Fanuc TP program (LS listing): UP022.LS

/PROG  UP022
/ATTR
OWNER		= MNEDITOR;
COMMENT		= "Soldadura Est.";
PROG_SIZE	= 11568;
CREATE		= DATE 23-07-08  TIME 22:50:50;
MODIFIED	= DATE 24-03-09  TIME 08:24:52;
FILE_NAME	= UP002;
VERSION		= 0;
LINE_COUNT	= 53;
MEMORY_SIZE	= 20152;
PROTECT		= READ_WRITE;
TCD:  STACK_SIZE	= 500,
      TASK_PRIORITY	= 50,
      TIME_SLICE	= 0,
      BUSY_LAMP_OFF	= 0,
      ABORT_REQUEST	= 0,
      PAUSE_REQUEST	= 0;
DEFAULT_GROUP	= 1,1,1,1,*;
CONTROL_CODE	= 00000001 00000000;
/APPL
/MN
   1:  UFRAME_NUM=1 ;
   2:  UTOOL_NUM=2 ;
   3:  PAYLOAD[2] ;
   4:J P[1] 100% CNT0 ACC100 TB    .10sec,P-SPS    ;
      1:  TC_ONLINE (ON) ;
      2:  DO[23]=OFF ;
      3:  TIMER[4]=RESET ;
      4:  TIMER[4]=START ;
      5:  CALL MAKRO050    ;
      6:  !Lib. de Herramientas ;
      7:  DO[80]=ON ;
      8:  DO[78]=OFF ;
      9:  DO[77]=ON ;
     10:  DO[75]=OFF ;
     11:  !Lib. de Anticolisiones ;
     12:  DO[41]=ON ;
     13:  DO[42]=ON ;
     14:  DO[43]=ON ;
     15:  DO[44]=ON ;
     16:  !Apagar Pos. Base ;
     17:  DO[15]=OFF ;
     18:  !Robot en Trayectoria ;
     19:  DO[16]=ON ;
     20:  !Basculante 1 en Pos. de Reposo ;
     21:  IF (!DI[842] AND DO[12]),CALL MAKRO072 ;
     22:  WAIT (M[96])    ;
     23:  WAIT (DI[23])    ;
     24:  DO[23]=(ON) ;
     25:  TC_ONLINE (M[1] AND M[30] AND M[31] AND M[34] AND M[35] AND M[95] AND M[96]) ;
       ------ ;
   5:J P[2] 100% CNT100 ACC100 TB   0.00sec,P-SPS    ;
      1:  TC_ONLINE (M[1] AND M[30] AND M[31] AND M[34] AND M[35] AND M[95] AND M[96]) ;
       ------ ;
   6:J P[3] 100% CNT100 ACC100 TB   0.00sec,P-SPS    ;
      1:  TC_ONLINE (M[1] AND M[30] AND M[31] AND M[34] AND M[35] AND M[95] AND M[96]) ;
       ------ ;
   7:J P[4] 100% CNT100 ACC100 TB   0.00sec,P-SPS    ;
      1:  TC_ONLINE (M[1] AND M[30] AND M[31] AND M[34] AND M[35] AND M[95] AND M[96]) ;
       ------ ;
   8:  !5QA802035b_017_R_PS_0031 ;
   9:  !Punto de Sol. No. 10094 ;
  10:J P[5] 100% CNT0 ACC100 TB    .10sec,P-SPS Offset,PR[11]    ;
      1:  TC_ONLINE (ON) ;
      2:  DO[23]=OFF ;
      3:  WAIT (!DI[16] AND DI[23])    ;
      4:  CALL VW_USER(Basic1,EZSP,Nr1,ProgNr=99, , ,S-Punkt=10094,Fzg_Typ=7,EIN/AUS=ON) ;
      5:  GO[2]=(R[197]) ;
      6:  WAIT (!DI[129] OR DI[26])    ;
      7:  CALL MAKRO080    ;
      8:  WAIT (DI[23])    ;
      9:  DO[23]=ON ;
     10:  TC_ONLINE (M[1] AND M[30] AND M[31] AND M[34] AND M[35] AND M[95] AND M[96]) ;
       ------ ;
  11:  !5QA802035b_017_R_PS_0029 ;
  12:  !Punto de Sol. No. 10095 ;
  13:J P[6] 100% CNT0 ACC100 TB    .10sec,P-SPS Offset,PR[11]    ;
      1:  TC_ONLINE (ON) ;
      2:  DO[23]=OFF ;
      3:  WAIT (!DI[16] AND DI[23])    ;
      4:  CALL VW_USER(Basic1,EZSP,Nr1,ProgNr=99, , ,S-Punkt=10095,Fzg_Typ=7,EIN/AUS=ON) ;
      5:  GO[2]=(R[197]) ;
      6:  WAIT (!DI[129] OR DI[26])    ;
      7:  CALL MAKRO080    ;
      8:  WAIT (DI[23])    ;
      9:  DO[23]=ON ;
     10:  TC_ONLINE (M[1] AND M[30] AND M[31] AND M[34] AND M[35] AND M[95] AND M[96]) ;
       ------ ;
  14:  !5QA802035b_017_R_PS_0028 ;
  15:  !Punto de Sol. No. 10096 ;
  16:J P[7] 100% CNT0 ACC100 TB    .10sec,P-SPS Offset,PR[11]    ;
      1:  TC_ONLINE (ON) ;
      2:  DO[23]=OFF ;
      3:  WAIT (!DI[16] AND DI[23])    ;
      4:  CALL VW_USER(Basic1,EZSP,Nr1,ProgNr=99, , ,S-Punkt=10096,Fzg_Typ=7,EIN/AUS=ON) ;
      5:  GO[2]=(R[197]) ;
      6:  WAIT (!DI[129] OR DI[26])    ;
      7:  CALL MAKRO080    ;
      8:  WAIT (DI[23])    ;
      9:  DO[23]=ON ;
     10:  TC_ONLINE (M[1] AND M[30] AND M[31] AND M[34] AND M[35] AND M[95] AND M[96]) ;
       ------ ;
  17:  !5QA802035b_017_R_PS_0027 ;
  18:  !Punto de Sol. No. 10097 ;
  19:J P[8] 100% CNT0 ACC100 TB    .10sec,P-SPS Offset,PR[11]    ;
      1:  TC_ONLINE (ON) ;
      2:  DO[23]=OFF ;
      3:  WAIT (!DI[16] AND DI[23])    ;
      4:  CALL VW_USER(Basic1,EZSP,Nr1,ProgNr=99, , ,S-Punkt=10097,Fzg_Typ=7,EIN/AUS=ON) ;
      5:  GO[2]=(R[197]) ;
      6:  WAIT (!DI[129] OR DI[26])    ;
      7:  CALL MAKRO080    ;
      8:  WAIT (DI[23])    ;
      9:  DO[23]=ON ;
     10:  TC_ONLINE (M[1] AND M[30] AND M[31] AND M[34] AND M[35] AND M[95] AND M[96]) ;
       ------ ;
  20:  !5QA802035b_017_R_PS_0026 ;
  21:  !Punto de Sol. No. 10098 ;
  22:J P[9] 100% CNT0 ACC100 TB    .10sec,P-SPS Offset,PR[11]    ;
      1:  TC_ONLINE (ON) ;
      2:  DO[23]=OFF ;
      3:  WAIT (!DI[16] AND DI[23])    ;
      4:  CALL VW_USER(Basic1,EZSP,Nr1,ProgNr=99, , ,S-Punkt=10098,Fzg_Typ=7,EIN/AUS=ON) ;
      5:  GO[2]=(R[197]) ;
      6:  WAIT (!DI[129] OR DI[26])    ;
      7:  CALL MAKRO080    ;
      8:  WAIT (DI[23])    ;
      9:  DO[23]=ON ;
     10:  TC_ONLINE (M[1] AND M[30] AND M[31] AND M[34] AND M[35] AND M[95] AND M[96]) ;
       ------ ;
  23:  !5QA802035b_017_R_PS_0025 ;
  24:  !Punto de Sol. No. 10099 ;
  25:J P[10] 100% CNT0 ACC100 TB    .10sec,P-SPS Offset,PR[11]    ;
      1:  TC_ONLINE (ON) ;
      2:  DO[23]=OFF ;
      3:  WAIT (!DI[16] AND DI[23])    ;
      4:  CALL VW_USER(Basic1,EZSP,Nr1,ProgNr=99, , ,S-Punkt=10099,Fzg_Typ=7,EIN/AUS=ON) ;
      5:  GO[2]=(R[197]) ;
      6:  WAIT (!DI[129] OR DI[26])    ;
      7:  CALL MAKRO080    ;
      8:  WAIT (DI[23])    ;
      9:  DO[23]=ON ;
     10:  TC_ONLINE (M[1] AND M[30] AND M[31] AND M[34] AND M[35] AND M[95] AND M[96]) ;
       ------ ;
  26:  !5QA802035b_017_R_PS_0001 ;
  27:  !Punto de Sol. No. 10100 ;
  28:J P[11] 100% CNT0 ACC100 TB    .10sec,P-SPS Offset,PR[11]    ;
      1:  TC_ONLINE (ON) ;
      2:  DO[23]=OFF ;
      3:  WAIT (!DI[16] AND DI[23])    ;
      4:  CALL VW_USER(Basic1,EZSP,Nr1,ProgNr=99, , ,S-Punkt=10100,Fzg_Typ=7,EIN/AUS=ON) ;
      5:  GO[2]=(R[197]) ;
      6:  WAIT (!DI[129] OR DI[26])    ;
      7:  CALL MAKRO080    ;
      8:  WAIT (DI[23])    ;
      9:  DO[23]=ON ;
     10:  TC_ONLINE (M[1] AND M[30] AND M[31] AND M[34] AND M[35] AND M[95] AND M[96]) ;
       ------ ;
  29:  !5QA802035b_017_R_PS_0019 ;
  30:  !Punto de Sol. No. 10101 ;
  31:J P[12] 100% CNT0 ACC100 TB    .10sec,P-SPS Offset,PR[11]    ;
      1:  TC_ONLINE (ON) ;
      2:  DO[23]=OFF ;
      3:  WAIT (!DI[16] AND DI[23])    ;
      4:  CALL VW_USER(Basic1,EZSP,Nr1,ProgNr=99, , ,S-Punkt=10101,Fzg_Typ=7,EIN/AUS=ON) ;
      5:  GO[2]=(R[197]) ;
      6:  WAIT (!DI[129] OR DI[26])    ;
      7:  CALL MAKRO080    ;
      8:  WAIT (DI[23])    ;
      9:  DO[23]=ON ;
     10:  TC_ONLINE (M[1] AND M[30] AND M[31] AND M[34] AND M[35] AND M[95] AND M[96]) ;
       ------ ;
  32:  !5QA802035b_017_R_PS_0020 ;
  33:  !Punto de Sol. No. 10102 ;
  34:J P[13] 100% CNT0 ACC100 TB    .10sec,P-SPS Offset,PR[11]    ;
      1:  TC_ONLINE (ON) ;
      2:  DO[23]=OFF ;
      3:  WAIT (!DI[16] AND DI[23])    ;
      4:  CALL VW_USER(Basic1,EZSP,Nr1,ProgNr=99, , ,S-Punkt=10102,Fzg_Typ=7,EIN/AUS=ON) ;
      5:  GO[2]=(R[197]) ;
      6:  WAIT (!DI[129] OR DI[26])    ;
      7:  CALL MAKRO080    ;
      8:  WAIT (DI[23])    ;
      9:  DO[23]=ON ;
     10:  TC_ONLINE (M[1] AND M[30] AND M[31] AND M[34] AND M[35] AND M[95] AND M[96]) ;
       ------ ;
  35:  !5QA802035b_017_R_PS_0023 ;
  36:  !Punto de Sol. No. 10103 ;
  37:J P[14] 100% CNT0 ACC100 TB    .10sec,P-SPS Offset,PR[11]    ;
      1:  TC_ONLINE (ON) ;
      2:  DO[23]=OFF ;
      3:  WAIT (!DI[16] AND DI[23])    ;
      4:  CALL VW_USER(Basic1,EZSP,Nr1,ProgNr=99, , ,S-Punkt=10103,Fzg_Typ=7,EIN/AUS=ON) ;
      5:  GO[2]=(R[197]) ;
      6:  WAIT (!DI[129] OR DI[26])    ;
      7:  CALL MAKRO080    ;
      8:  WAIT (DI[23])    ;
      9:  DO[23]=ON ;
     10:  TC_ONLINE (M[1] AND M[30] AND M[31] AND M[34] AND M[35] AND M[95] AND M[96]) ;
       ------ ;
  38:  !5QA802035b_017_R_PS_0002 ;
  39:  !Punto de Sol. No. 10104 ;
  40:J P[15] 100% CNT0 ACC100 TB    .10sec,P-SPS Offset,PR[11]    ;
      1:  TC_ONLINE (ON) ;
      2:  DO[23]=OFF ;
      3:  WAIT (!DI[16] AND DI[23])    ;
      4:  CALL VW_USER(Basic1,EZSP,Nr1,ProgNr=99, , ,S-Punkt=10104,Fzg_Typ=7,EIN/AUS=ON) ;
      5:  GO[2]=(R[197]) ;
      6:  WAIT (!DI[129] OR DI[26])    ;
      7:  CALL MAKRO080    ;
      8:  WAIT (DI[23])    ;
      9:  DO[23]=ON ;
     10:  TC_ONLINE (M[1] AND M[30] AND M[31] AND M[34] AND M[35] AND M[95] AND M[96]) ;
       ------ ;
  41:J P[16] 100% CNT100 ACC100 TB   0.00sec,P-SPS    ;
      1:  TC_ONLINE (M[1] AND M[30] AND M[31] AND M[34] AND M[35] AND M[95] AND M[96]) ;
       ------ ;
  42:J P[17] 100% CNT100 ACC100 TB   0.00sec,P-SPS    ;
      1:  TC_ONLINE (M[1] AND M[30] AND M[31] AND M[34] AND M[35] AND M[95] AND M[96]) ;
       ------ ;
  43:  !5QA802035b_017_R_PS_0007 ;
  44:  !Punto de Sol. No. 10105 ;
  45:J P[18] 100% CNT0 ACC100 TB    .10sec,P-SPS Offset,PR[11]    ;
      1:  TC_ONLINE (ON) ;
      2:  DO[23]=OFF ;
      3:  WAIT (!DI[16] AND DI[23])    ;
      4:  CALL VW_USER(Basic1,EZSP,Nr1,ProgNr=99, , ,S-Punkt=10105,Fzg_Typ=7,EIN/AUS=ON) ;
      5:  GO[2]=(R[197]) ;
      6:  WAIT (!DI[129] OR DI[26])    ;
      7:  CALL MAKRO080    ;
      8:  WAIT (DI[23])    ;
      9:  DO[23]=ON ;
     10:  TC_ONLINE (M[1] AND M[30] AND M[31] AND M[34] AND M[35] AND M[95] AND M[96]) ;
       ------ ;
  46:  !5QA802035_017_R_PS_0008 ;
  47:  !Punto de Sol. No. 10106 ;
  48:  !Fin de Trabajo 2 ;
  49:J P[19] 100% CNT0 ACC100 TB    .10sec,P-SPS Offset,PR[11]    ;
      1:  TC_ONLINE (ON) ;
      2:  DO[23]=OFF ;
      3:  WAIT (!DI[16] AND DI[23])    ;
      4:  CALL VW_USER(Basic1,EZSP,Nr1,ProgNr=99, , ,S-Punkt=10106,Fzg_Typ=7,EIN/AUS=ON) ;
      5:  GO[2]=(R[197]) ;
      6:  WAIT (!DI[129] OR DI[26])    ;
      7:  CALL MAKRO080    ;
      8:  IF (!DI[145] AND !DI[129]),CALL MAKRO002 ;
      9:  WAIT (DI[23])    ;
     10:  DO[23]=ON ;
     11:  TC_ONLINE (M[1] AND M[30] AND M[31] AND M[34] AND M[35] AND M[95] AND M[96]) ;
       ------ ;
  50:J P[20] 100% CNT100 ACC100 TB   0.00sec,P-SPS    ;
      1:  TC_ONLINE (M[1] AND M[30] AND M[31] AND M[34] AND M[35] AND M[95] AND M[96]) ;
       ------ ;
  51:J P[21] 100% CNT100 ACC100 TB   0.00sec,P-SPS    ;
      1:  TC_ONLINE (M[1] AND M[30] AND M[31] AND M[34] AND M[35] AND M[95] AND M[96]) ;
       ------ ;
  52:J P[22] 100% CNT100 ACC100 TB   0.00sec,P-SPS    ;
      1:  TC_ONLINE (M[1] AND M[30] AND M[31] AND M[34] AND M[35] AND M[95] AND M[96]) ;
       ------ ;
  53:J P[23] 100% CNT0 ACC100 TB    .10sec,P-SPS    ;
      1:  TC_ONLINE (ON) ;
      2:  DO[23]=OFF ;
      3:  TIMER[4]=STOP ;
      4:  WAIT (DI[23])    ;
      5:  CALL VW_USER(Basic1,EZSP,Nr1,ProgNr=31, , ,S-Punkt=31, ,EIN/AUS=1) ;
      6:  DO[23]=ON ;
      7:  TC_ONLINE (M[1] AND M[30] AND M[31] AND M[34] AND M[35] AND M[95] AND M[96]) ;
       ------ ;
/POS
P[1]{
   GP1:
	UF : 1, UT : 2,		CONFIG : 'N U T, 0, 0, 0',
	RX = -1379.596  mm,	RY =   331.266  mm,	RZ =  -697.223  mm,
	RW =    44.990 deg,	RP =   -45.000 deg,	RR =    90.014 deg
   GP2:
	UF : 1, UT : 2,
	J1=   100.000  mm
   GP3:
	UF : 1, UT : 2,
	J1=     0.000  mm
   GP4:
	UF : 1, UT : 2,
	J1=     0.000  mm
};
P[2]{
   GP1:
	UF : 1, UT : 2,		CONFIG : 'N U T, 0, 0, 0',
	RX =   559.428  mm,	RY =  -243.349  mm,	RZ = -1295.960  mm,
	RW =    -2.225 deg,	RP =    -4.071 deg,	RR =   169.322 deg
   GP2:
	UF : 1, UT : 2,
	J1=   100.000  mm
   GP3:
	UF : 1, UT : 2,
	J1=     0.000  mm
   GP4:
	UF : 1, UT : 2,
	J1=     0.000  mm
};
P[3]{
   GP1:
	UF : 1, UT : 2,		CONFIG : 'N U T, 0, 0, 0',
	RX =  -281.806  mm,	RY =  -499.725  mm,	RZ =   -17.895  mm,
	RW =    37.746 deg,	RP =    -1.264 deg,	RR =    94.148 deg
   GP2:
	UF : 1, UT : 2,
	J1=   100.000  mm
   GP3:
	UF : 1, UT : 2,
	J1=     0.000  mm
   GP4:
	UF : 1, UT : 2,
	J1=     0.000  mm
};
P[4]{
   GP1:
	UF : 1, UT : 2,		CONFIG : 'N U T, 0, 0, 0',
	RX =  -159.437  mm,	RY =  -499.603  mm,	RZ =   140.422  mm,
	RW =    37.745 deg,	RP =    -1.264 deg,	RR =    94.148 deg
   GP2:
	UF : 1, UT : 2,
	J1=   100.000  mm
   GP3:
	UF : 1, UT : 2,
	J1=     0.000  mm
   GP4:
	UF : 1, UT : 2,
	J1=     0.000  mm
};
P[5]{
   GP1:
	UF : 1, UT : 2,		CONFIG : 'N U T, 0, 0, 0',
	RX =  -162.152  mm,	RY =  -495.825  mm,	RZ =   145.300  mm,
	RW =    37.763 deg,	RP =     -.671 deg,	RR =    93.138 deg
   GP2:
	UF : 1, UT : 2,
	J1=    24.250  mm
   GP3:
	UF : 1, UT : 2,
	J1=     0.000  mm
   GP4:
	UF : 1, UT : 2,
	J1=     0.000  mm
};
P[6]{
   GP1:
	UF : 1, UT : 2,		CONFIG : 'N U T, 0, 0, 0',
	RX =  -235.073  mm,	RY =  -497.076  mm,	RZ =   148.662  mm,
	RW =    37.879 deg,	RP =    -3.500 deg,	RR =    88.275 deg
   GP2:
	UF : 1, UT : 2,
	J1=    24.956  mm
   GP3:
	UF : 1, UT : 2,
	J1=     0.000  mm
   GP4:
	UF : 1, UT : 2,
	J1=     0.000  mm
};
P[7]{
   GP1:
	UF : 1, UT : 2,		CONFIG : 'N U T, 0, 0, 0',
	RX =  -268.901  mm,	RY =  -495.720  mm,	RZ =   148.758  mm,
	RW =    38.051 deg,	RP =    -3.683 deg,	RR =    86.764 deg
   GP2:
	UF : 1, UT : 2,
	J1=    27.692  mm
   GP3:
	UF : 1, UT : 2,
	J1=     0.000  mm
   GP4:
	UF : 1, UT : 2,
	J1=     0.000  mm
};
P[8]{
   GP1:
	UF : 1, UT : 2,		CONFIG : 'N U T, 0, 0, 0',
	RX =  -306.980  mm,	RY =  -494.487  mm,	RZ =   150.141  mm,
	RW =    37.909 deg,	RP =    -4.476 deg,	RR =    86.639 deg
   GP2:
	UF : 1, UT : 2,
	J1=    27.222  mm
   GP3:
	UF : 1, UT : 2,
	J1=     0.000  mm
   GP4:
	UF : 1, UT : 2,
	J1=     0.000  mm
};
P[9]{
   GP1:
	UF : 1, UT : 2,		CONFIG : 'N U T, 0, 0, 0',
	RX =  -338.044  mm,	RY =  -493.552  mm,	RZ =   151.355  mm,
	RW =    37.814 deg,	RP =    -3.392 deg,	RR =    87.875 deg
   GP2:
	UF : 1, UT : 2,
	J1=    29.615  mm
   GP3:
	UF : 1, UT : 2,
	J1=     0.000  mm
   GP4:
	UF : 1, UT : 2,
	J1=     0.000  mm
};
P[10]{
   GP1:
	UF : 1, UT : 2,		CONFIG : 'N U T, 0, 0, 0',
	RX =  -373.481  mm,	RY =  -496.493  mm,	RZ =   150.285  mm,
	RW =    37.504 deg,	RP =    -2.638 deg,	RR =    98.581 deg
   GP2:
	UF : 1, UT : 2,
	J1=    29.848  mm
   GP3:
	UF : 1, UT : 2,
	J1=     0.000  mm
   GP4:
	UF : 1, UT : 2,
	J1=     0.000  mm
};
P[11]{
   GP1:
	UF : 1, UT : 2,		CONFIG : 'N U T, 0, 0, 0',
	RX =  -411.180  mm,	RY =  -513.262  mm,	RZ =   150.125  mm,
	RW =    35.821 deg,	RP =    -2.194 deg,	RR =   116.945 deg
   GP2:
	UF : 1, UT : 2,
	J1=    27.096  mm
   GP3:
	UF : 1, UT : 2,
	J1=     0.000  mm
   GP4:
	UF : 1, UT : 2,
	J1=     0.000  mm
};
P[12]{
   GP1:
	UF : 1, UT : 2,		CONFIG : 'N U T, 0, 0, 0',
	RX =  -443.061  mm,	RY =  -521.242  mm,	RZ =   152.453  mm,
	RW =    39.674 deg,	RP =     1.537 deg,	RR =    85.624 deg
   GP2:
	UF : 1, UT : 2,
	J1=    25.000  mm
   GP3:
	UF : 1, UT : 2,
	J1=     0.000  mm
   GP4:
	UF : 1, UT : 2,
	J1=     0.000  mm
};
P[13]{
   GP1:
	UF : 1, UT : 2,		CONFIG : 'N U T, 0, 0, 0',
	RX =  -468.095  mm,	RY =  -523.751  mm,	RZ =   154.064  mm,
	RW =    41.322 deg,	RP =      .078 deg,	RR =    87.815 deg
   GP2:
	UF : 1, UT : 2,
	J1=    25.984  mm
   GP3:
	UF : 1, UT : 2,
	J1=     0.000  mm
   GP4:
	UF : 1, UT : 2,
	J1=     0.000  mm
};
P[14]{
   GP1:
	UF : 1, UT : 2,		CONFIG : 'N U T, 0, 0, 0',
	RX =  -567.321  mm,	RY =  -526.172  mm,	RZ =   153.295  mm,
	RW =    40.497 deg,	RP =     -.144 deg,	RR =    89.127 deg
   GP2:
	UF : 1, UT : 2,
	J1=    26.768  mm
   GP3:
	UF : 1, UT : 2,
	J1=     0.000  mm
   GP4:
	UF : 1, UT : 2,
	J1=     0.000  mm
};
P[15]{
   GP1:
	UF : 1, UT : 2,		CONFIG : 'N U T, 0, 0, 0',
	RX =  -621.541  mm,	RY =  -529.083  mm,	RZ =   154.560  mm,
	RW =    39.632 deg,	RP =      .959 deg,	RR =    87.452 deg
   GP2:
	UF : 1, UT : 2,
	J1=    33.566  mm
   GP3:
	UF : 1, UT : 2,
	J1=     0.000  mm
   GP4:
	UF : 1, UT : 2,
	J1=     0.000  mm
};
P[16]{
   GP1:
	UF : 1, UT : 2,		CONFIG : 'N U T, 0, 0, 0',
	RX =  -567.802  mm,	RY =  -526.963  mm,	RZ =   150.972  mm,
	RW =    41.336 deg,	RP =     0.000 deg,	RR =    90.000 deg
   GP2:
	UF : 1, UT : 2,
	J1=   180.000  mm
   GP3:
	UF : 1, UT : 2,
	J1=     0.000  mm
   GP4:
	UF : 1, UT : 2,
	J1=     0.000  mm
};
P[17]{
   GP1:
	UF : 1, UT : 2,		CONFIG : 'N U T, 0, 0, 0',
	RX =  -526.369  mm,	RY =  -526.984  mm,	RZ =   294.289  mm,
	RW =    41.336 deg,	RP =     -.002 deg,	RR =    89.997 deg
   GP2:
	UF : 1, UT : 2,
	J1=   180.000  mm
   GP3:
	UF : 1, UT : 2,
	J1=     0.000  mm
   GP4:
	UF : 1, UT : 2,
	J1=     0.000  mm
};
P[18]{
   GP1:
	UF : 1, UT : 2,		CONFIG : 'N U T, 0, 0, 0',
	RX =  -519.912  mm,	RY =  -520.462  mm,	RZ =   291.943  mm,
	RW =    41.344 deg,	RP =      .002 deg,	RR =    89.996 deg
   GP2:
	UF : 1, UT : 2,
	J1=    30.200  mm
   GP3:
	UF : 1, UT : 2,
	J1=     0.000  mm
   GP4:
	UF : 1, UT : 2,
	J1=     0.000  mm
};
P[19]{
   GP1:
	UF : 1, UT : 2,		CONFIG : 'N U T, 0, 0, 0',
	RX =  -486.324  mm,	RY =  -520.011  mm,	RZ =   293.059  mm,
	RW =    41.339 deg,	RP =     -.000 deg,	RR =    89.995 deg
   GP2:
	UF : 1, UT : 2,
	J1=    32.500  mm
   GP3:
	UF : 1, UT : 2,
	J1=     0.000  mm
   GP4:
	UF : 1, UT : 2,
	J1=     0.000  mm
};
P[20]{
   GP1:
	UF : 1, UT : 2,		CONFIG : 'N U T, 0, 0, 0',
	RX =  -498.582  mm,	RY =  -520.026  mm,	RZ =   294.290  mm,
	RW =    41.336 deg,	RP =     -.002 deg,	RR =    89.997 deg
   GP2:
	UF : 1, UT : 2,
	J1=   180.000  mm
   GP3:
	UF : 1, UT : 2,
	J1=     0.000  mm
   GP4:
	UF : 1, UT : 2,
	J1=     0.000  mm
};
P[21]{
   GP1:
	UF : 1, UT : 2,		CONFIG : 'N U T, 0, 0, 0',
	RX =  -162.032  mm,	RY =  -564.996  mm,	RZ =  -172.337  mm,
	RW =    16.262 deg,	RP =     -.000 deg,	RR =    90.003 deg
   GP2:
	UF : 1, UT : 2,
	J1=   180.000  mm
   GP3:
	UF : 1, UT : 2,
	J1=     0.000  mm
   GP4:
	UF : 1, UT : 2,
	J1=     0.000  mm
};
P[22]{
   GP1:
	UF : 1, UT : 2,		CONFIG : 'N U T, 0, 0, 0',
	RX =   638.674  mm,	RY =  -300.483  mm,	RZ = -1271.750  mm,
	RW =      .017 deg,	RP =    -1.407 deg,	RR =   172.462 deg
   GP2:
	UF : 1, UT : 2,
	J1=   100.000  mm
   GP3:
	UF : 1, UT : 2,
	J1=     0.000  mm
   GP4:
	UF : 1, UT : 2,
	J1=     0.000  mm
};
P[23]{
   GP1:
	UF : 1, UT : 2,		CONFIG : 'N U T, 0, 0, 0',
	RX = -1379.596  mm,	RY =   331.265  mm,	RZ =  -697.223  mm,
	RW =    44.990 deg,	RP =   -45.000 deg,	RR =    90.014 deg
   GP2:
	UF : 1, UT : 2,
	J1=   100.000  mm
   GP3:
	UF : 1, UT : 2,
	J1=     0.000  mm
   GP4:
	UF : 1, UT : 2,
	J1=     0.000  mm
};
/END
